Staubli VAL3: onF8Event.pgx

program onF8Event(bool& x_bSave[])
  local trsf l_tEmpty
  local num l_nSize
begin
  // look if the bButton is enable
  if bButton[7]
    //
    l_tEmpty={0,0,0,0,0,0}
    call tcp:new(l_tEmpty)
    call tcp:getSize(l_nSize)
    nIndexTool=l_nSize-1
    // refresh and modify the name
    call buildList()
    call refreshStatic()
    nIndex=0
    sEvent=""
    call editTool(l_tEmpty)
    logMsg("[VALlaser] INTERFACE:Insert new tool at index: "+toString("",l_nSize))
    x_bSave=true
  endIf
end
